Fanuc KAREL source: KO00140.KL

PROGRAM KO00140
%NOLOCKGROUP
VAR
  R: REAL
  CFG: CONFIG
  OUT: XYZWPR
  N: ARRAY[2] OF SHORT
BEGIN
  N[1] = 1
  R = 2.0
  CFG.CFG_FLIP = TRUE
  OUT = POS(R, R, N[1], R, R, R, CFG)
END KO00140
